Staubli VAL3: page_simulation.dtx

num nEvent
num nIndex
num nKey
public num nPage
num nPoint
num nRefresh = 1
num nSelect
num nTime = 1.5
public num nToSuperV
num nRoundStepping = 25
num nMoveId
string sEvent
public string sItems
string sList
string sMenu
string sMessage
string sTrajName
string sMenu8[8]
bool bButton[8]
bool bMoveToPoint
bool bShowMessage
bool bShowStatus
bool bStepping
mdesc nom_speed = {accel=50, vel=50, decel=50, tmax=999, rmax=999, blend=off}
